FUNCTION_BLOCK PI_LEVEL_CONTROLLER (* PI level controller with anti-windup, manual tracking, and diagnostics *)
  (* Standard: 61499-2 *)
  (* Version 1.0, 2026-07-24, Guilherme *)
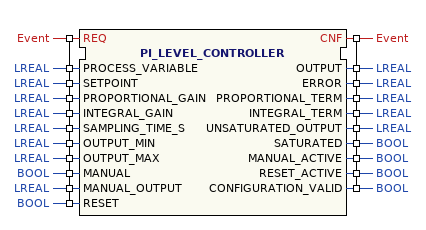
  EVENT_INPUT
    REQ WITH PROCESS_VARIABLE, SETPOINT, PROPORTIONAL_GAIN, INTEGRAL_GAIN, SAMPLING_TIME_S, OUTPUT_MIN, OUTPUT_MAX, MANUAL, MANUAL_OUTPUT, RESET; (* Execute one PI controller cycle *)
  END_EVENT
  EVENT_OUTPUT
    CNF WITH OUTPUT, ERROR, PROPORTIONAL_TERM, INTEGRAL_TERM, UNSATURATED_OUTPUT, SATURATED, MANUAL_ACTIVE, RESET_ACTIVE, CONFIGURATION_VALID; (* Controller cycle completed *)
  END_EVENT
  VAR_INPUT
    PROCESS_VARIABLE : LREAL; (* Measured process level *)
    SETPOINT : LREAL; (* Desired process level *)
    PROPORTIONAL_GAIN : LREAL; (* Proportional gain *)
    INTEGRAL_GAIN : LREAL; (* Integral gain *)
    SAMPLING_TIME_S : LREAL; (* Controller sampling time in seconds *)
    OUTPUT_MIN : LREAL; (* Minimum controller output *)
    OUTPUT_MAX : LREAL; (* Maximum controller output *)
    MANUAL : BOOL; (* Enable manual mode *)
    MANUAL_OUTPUT : LREAL; (* Requested output in manual mode *)
    RESET : BOOL; (* Apply deterministic reset behavior *)
  END_VAR
  VAR_OUTPUT
    OUTPUT : LREAL; (* Saturated controller output *)
    ERROR : LREAL; (* Setpoint minus process variable *)
    PROPORTIONAL_TERM : LREAL; (* Proportional contribution *)
    INTEGRAL_TERM : LREAL; (* Stored integral contribution *)
    UNSATURATED_OUTPUT : LREAL; (* Controller output before clamping *)
    SATURATED : BOOL; (* Output or manual command was clamped *)
    MANUAL_ACTIVE : BOOL; (* Controller cycle executed in manual mode *)
    RESET_ACTIVE : BOOL; (* Controller cycle executed reset behavior *)
    CONFIGURATION_VALID : BOOL; (* Sampling time and output limits are valid *)
  END_VAR
  VAR
    integral_term_internal : LREAL := 0.0; (* Stored integral contribution *)
    manual_was_active : BOOL := FALSE; (* Previous cycle used manual mode *)
    integral_increment : LREAL := 0.0; (* Candidate integral change *)
    candidate_integral : LREAL := 0.0; (* Candidate integral contribution *)
    candidate_unsaturated_output : LREAL := 0.0; (* Candidate output before anti-windup decision *)
    clamped_manual_output : LREAL := 0.0; (* Manual command after output limits *)
  END_VAR
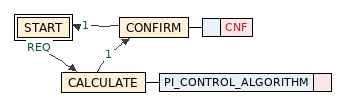
  EC_STATES
    START; (* Initial state *)
    CALCULATE : PI_CONTROL_ALGORITHM; (* Execute the PI algorithm *)
    CONFIRM : -> CNF; (* Publish controller outputs *)
  END_STATES
  EC_TRANSITIONS
    START TO CALCULATE := REQ;
    CALCULATE TO CONFIRM := 1;
    CONFIRM TO START := 1;
  END_TRANSITIONS
  ALGORITHM PI_CONTROL_ALGORITHM IN ST: (* Positional PI controller with conditional anti-windup and manual tracking *)
ERROR := SETPOINT - PROCESS_VARIABLE;
PROPORTIONAL_TERM := PROPORTIONAL_GAIN * ERROR;

CONFIGURATION_VALID :=
    (SAMPLING_TIME_S > 0.0)
    AND
    (OUTPUT_MIN < OUTPUT_MAX);

IF NOT CONFIGURATION_VALID THEN
    integral_term_internal := 0.0;
    manual_was_active := FALSE;

    OUTPUT := 0.0;
    INTEGRAL_TERM := 0.0;
    UNSATURATED_OUTPUT := 0.0;
    SATURATED := FALSE;
    MANUAL_ACTIVE := FALSE;
    RESET_ACTIVE := FALSE;

ELSIF RESET THEN
    integral_term_internal := 0.0;
    manual_was_active := FALSE;

    OUTPUT := 0.0;

    IF OUTPUT > OUTPUT_MAX THEN
        OUTPUT := OUTPUT_MAX;
    ELSIF OUTPUT < OUTPUT_MIN THEN
        OUTPUT := OUTPUT_MIN;
    END_IF;

    INTEGRAL_TERM := 0.0;
    UNSATURATED_OUTPUT := OUTPUT;
    SATURATED := FALSE;
    MANUAL_ACTIVE := MANUAL;
    RESET_ACTIVE := TRUE;

ELSIF MANUAL THEN
    clamped_manual_output := MANUAL_OUTPUT;

    IF clamped_manual_output > OUTPUT_MAX THEN
        clamped_manual_output := OUTPUT_MAX;
    ELSIF clamped_manual_output < OUTPUT_MIN THEN
        clamped_manual_output := OUTPUT_MIN;
    END_IF;

    OUTPUT := clamped_manual_output;
    integral_term_internal := OUTPUT - PROPORTIONAL_TERM;

    INTEGRAL_TERM := integral_term_internal;
    UNSATURATED_OUTPUT := OUTPUT;
    SATURATED := OUTPUT <> MANUAL_OUTPUT;
    MANUAL_ACTIVE := TRUE;
    RESET_ACTIVE := FALSE;
    manual_was_active := TRUE;

ELSE
    IF manual_was_active THEN
        manual_was_active := FALSE;
    ELSE
        integral_increment :=
            INTEGRAL_GAIN
            * ERROR
            * SAMPLING_TIME_S;

        candidate_integral :=
            integral_term_internal
            + integral_increment;

        candidate_unsaturated_output :=
            PROPORTIONAL_TERM
            + candidate_integral;

        IF NOT (
            (
                candidate_unsaturated_output > OUTPUT_MAX
                AND
                integral_increment > 0.0
            )
            OR
            (
                candidate_unsaturated_output < OUTPUT_MIN
                AND
                integral_increment < 0.0
            )
        ) THEN
            integral_term_internal :=
                candidate_integral;
        END_IF;
    END_IF;

    INTEGRAL_TERM := integral_term_internal;

    UNSATURATED_OUTPUT :=
        PROPORTIONAL_TERM
        + INTEGRAL_TERM;

    OUTPUT := UNSATURATED_OUTPUT;

    IF OUTPUT > OUTPUT_MAX THEN
        OUTPUT := OUTPUT_MAX;
    ELSIF OUTPUT < OUTPUT_MIN THEN
        OUTPUT := OUTPUT_MIN;
    END_IF;

    SATURATED := OUTPUT <> UNSATURATED_OUTPUT;
    MANUAL_ACTIVE := FALSE;
    RESET_ACTIVE := FALSE;
END_IF;
  END_ALGORITHM
END_FUNCTION_BLOCK
